PROGRAM P_Demo_F_BA_ByteCmp
VAR
    argPValue                      : PVOID                          := 0; // pValue
    argNSize                       : UXINT                         ; // nSize
    argNCompare                    : BYTE                           := 0; // nCompare
    fnReturn                       : DINT; // 返回值
END_VAR

// =============================================================================
// Tc3_BA2_Common.F_BA_ByteCmp 演示程序
// =============================================================================
// 场景：检查一段 buffer 是否全是 `0x00`（未初始化检测）或全是 `0xFF`（擦除标志位）。
//
// 价值：比 `MEMCMP` 更轻量（不用第二个 buffer），适合"全 0 / 全 FF / 全单字节模式"快速判定。
//
// 验证：登录 PLC 后，按例程内变量在线写值；监视输出 / 返回值，结合 §1 功能
//       简述的预期行为对照（详见配套 .md 文档 §7 业务场景）。
//
// 验证步骤：
//   1. 右键 PLC 项目下 POUs 文件夹 → Add → Existing Item → 选本 .TcPOU 文件
//   2. 引用 Tc3_BA2_Common（References → Add library）
//   3. 编译 → 登录 → 运行；按上方『验证』指引在线写值观察
// =============================================================================

fnReturn := F_BA_ByteCmp(
    pValue                   := argPValue,
    nSize                    := argNSize,
    nCompare                 := argNCompare
);

END_PROGRAM

(* stored: Version 1.1.0.1, ProductVersion 3.1.4024.5
   POU P_Demo_F_BA_ByteCmp: Id {c7631e9b-c7fa-578b-ab48-0336cbc04141}, SpecialFunc None *)
